// TwinCAT 3 PLC project TcoData
// Title: TcoData
// Company: Vortex.Library
// ProjectVersion: 0.6.0.913
// ProgramVersion: 3.1.4023.0
// libraries:
//   Tc2_Standard, * (Beckhoff Automation GmbH)
//   Tc2_System, * (Beckhoff Automation GmbH)
//   Tc3_Module, * (Beckhoff Automation GmbH)
//   TcoCore, 0.6.0.913 (Vortex.Library)
// project tree:
//   / PlcTask.TcTTO
//   POUs/Data/ TcoEntity.TcDUT, ITcoCrud.TcIO, TcoDataExchange.TcPOU, TcoDataTask.TcPOU, TcoExistsTask.TcPOU
//   POUs/ MAIN.TcPOU, MainContext.TcPOU
// real-time tasks:
//   TASK PlcTask: cycle T#10ms, priority 20, ADS port 350

CONFIGURATION TcoData
    RESOURCE PLC ON TwinCAT3
        TASK PlcTask(INTERVAL := T#10ms, PRIORITY := 20);
        PROGRAM MAIN WITH PlcTask : MAIN;
    END_RESOURCE
END_CONFIGURATION

// ---- POUs/Data/TcoEntity.TcDUT
(*~
    <docu>
        <summary>
            Base strucure of any data entity used in TcoDataExchange.
            <remarks>
                   <note type="information">
                    Inxton is required for this feature to work.
                   </note>
            </remarks>
        </summary>

        <example>
            [!code-pas[Declarations](~/../TcOpen/src/TcoData/src/XAE/XAE/TcoDataTests/POUs/Examples/SandboxData.TcDUT?name=SandboxData)]
        </example>
    </docu>
~*)
TYPE TcoEntity EXTENDS TcoCore.TcoStruct :
STRUCT
    {attribute wpf [Container(Layout.Stack)]}
    {attribute addProperty Name "<#ID#>"}
    {attribute clr [RenderIgnore("Control", "ShadowControl", "ControlSlim", "ShadowControlSlim")]}
    _EntityId : STRING(254);
END_STRUCT
END_TYPE

// ---- POUs/Data/ITcoCrud.TcIO
INTERFACE ITcoCrud

METHOD Create : TcoCore.ITcoTaskStatus
VAR_INPUT
	Identifier : STRING(255);
END_VAR
END_METHOD

METHOD Delete : TcoCore.ITcoTaskStatus
VAR_INPUT
	Identifier : STRING(255);
END_VAR
END_METHOD

METHOD Read : TcoCore.ITcoTaskStatus
VAR_INPUT
	Identifier : STRING(255);
END_VAR
END_METHOD

METHOD Update : TcoCore.ITcoTaskStatus
VAR_INPUT
	Identifier : STRING(255);
END_VAR
END_METHOD

END_INTERFACE

// ---- POUs/MAIN.TcPOU
PROGRAM INTERNAL MAIN
VAR
    Context : MainContext;
END_VAR

END_PROGRAM

// ---- POUs/MainContext.TcPOU
FUNCTION_BLOCK INTERNAL MainContext EXTENDS TcoCore.TcoContext
VAR
    fbProcessDataManger : TcoDataExchange(THIS^);
    test : TcoEntity;
END_VAR

(*~
    <docu>
        <summary>
            Main method of the TcoContext. This is the entry point of any control logic that belongs to this context.
            The call of this method is ensured by calling the <c>InstanceName.Run()</c> method, and it must not be called explicitly.
            This method is abstract, and it must be overridden in derived block.
        </summary>
    </docu>
~*)
METHOD PROTECTED Main
END_METHOD

END_FUNCTION_BLOCK

// ---- POUs/Data/TcoDataExchange.TcPOU
(*~
    <docu>
        <summary>
            Provides a mechanism to exchange data between PLC and an arbitrary data repository.
            TcoDataExchange support Create, Read, Update, Delete (CRUD) operations and some additional
            functions.
            TcoDataExchange **operates by convention on data member named `_data`** declared in the function block.
            The `_data` member must be of type that extends `TcoData.TcoEntity`.
            TcoDataEchange must be then inizialized in the higher level application where the repository
            and remote data exchange is configured.
            <remarks>
                   <note type="information">
                    Inxton is required for this feature to work.
                   </note>
            </remarks>
        </summary>

        <example>
            [!code-pas[Declarations](~/../TcOpen/src/TcoData/src/XAE/XAE/TcoDataTests/POUs/Examples/TcoDataManager.TcPOU?name=DataManagerDeclarations)]
            [!code-pas[SuperCall](~/../TcOpen/src/TcoData/src/XAE/XAE/TcoDataTests/POUs/Examples/TcoDataManager.TcPOU?name=DataManagerSuperCall)]
            [!code-pas[Data](~/../TcOpen/src/TcoData/src/XAE/XAE/TcoDataTests/POUs/Examples/SandboxData.TcDUT?name=SandboxData)]
            [!code-csharp[Main](~/../TcOpen/src/TcoData/tests/TcoDataExamples.Tests/SandboxContextTests.cs?name=RepositoryInitialization)]
        </example>
    </docu>
~*)
FUNCTION_BLOCK TcoDataExchange EXTENDS TcoCore.TcoObject IMPLEMENTS ITcoCrud
VAR
    (*~
        <docu>
            <summary>
                Instance of task that `creates` the entry into repository.
            </summary>
        </docu>
    ~*)
    _createTask : TcoDataTask(THIS^);
    (*~
        <docu>
            <summary>
                Instance of task that `reads` the entry from repository.
            </summary>
        </docu>
    ~*)
    _readTask : TcoDataTask(THIS^);
    (*~
        <docu>
            <summary>
                Instance of task that `updates` record in the repository.
            </summary>
        </docu>
    ~*)
    _updateTask : TcoDataTask(THIS^);
    (*~
        <docu>
            <summary>
                Instance of task that `deletes` record from the repository.
            </summary>
        </docu>
    ~*)
    _deleteTask : TcoDataTask(THIS^);
    (*~
        <docu>
            <summary>
                Instance of task that `check for existence` of a record with an `id` in the repository.
            </summary>
        </docu>
    ~*)
    _idExistsTask : TcoExistsTask(THIS^);
    (*~
        <docu>
            <summary>
                Instance of task that `creates inexisting or updates existing` record in the repository.
            </summary>
        </docu>
    ~*)
    _createOrUpdateTask : TcoDataTask(THIS^);
END_VAR

_createTask();
_readTask();
_updateTask();
_deleteTask();
_idExistsTask();
_createOrUpdateTask();

(*~
    <docu>
        <summary>
            Creates new entry in the Repository from `_data` member of this `TcoDataExchange`.
            <remarks>
                   <note type="information">
                    Inxton is required for this feature to work.
                   </note>
            </remarks>
        </summary>

        <example>
            [!code-pas[Main](~/../TcOpen/src/TcoData/src/XAE/XAE/TcoDataTests/POUs/Examples/SandboxContext.TcPOU?name=CreateCodeExample)]
        </example>
    </docu>
~*)
METHOD Create : TcoCore.ITcoTaskStatus
VAR_INPUT
    (*~
    <docu>
        <summary>
            Identifier of the data entry to be created in the repository.
        </summary>

    </docu>
    ~*)
    Identifier : STRING(255);
END_VAR
Create := _createTask.WithId(Identifier).Invoke();
THIS^.Messenger.Build().Append('<#Creating data item with id:#> ').Append(Identifier).As().AsTrace();
END_METHOD

(*~
    <docu>
        <summary>
            Creates or updates new entry in the Repository from `_data` member of this `TcoDataExchange`.
            <remarks>
                   <note type="information">
                    Inxton is required for this feature to work.
                   </note>
            </remarks>
        </summary>

        <example>
            [!code-pas[Main](~/../TcOpen/src/TcoData/src/XAE/XAE/TcoDataTests/POUs/Examples/SandboxContext.TcPOU?name=CreateOrUpdateCodeExample)]
        </example>
    </docu>
~*)
METHOD CreateOrUpdate : TcoCore.ITcoTaskStatus
VAR_INPUT
    (*~
        <docu>
            <summary>
                Identifier of the data entry to be created or updated in the repository.
            </summary>

        </docu>
    ~*)
    Identifier : STRING(255);
END_VAR
CreateOrUpdate := _createOrUpdateTask.WithId(Identifier).Invoke();
THIS^.Messenger.Build().Append('<#Creating or updating data item with id:#> ').Append(Identifier).As().AsTrace();
END_METHOD

(*~
    <docu>
        <summary>
            Deletes an item from the repository.
            <remarks>
                   <note type="information">
                    Inxton is required for this feature to work.
                   </note>
            </remarks>
        </summary>

        <example>
            [!code-pas[Main](~/../TcOpen/src/TcoData/src/XAE/XAE/TcoDataTests/POUs/Examples/SandboxContext.TcPOU?name=DeleteCodeExample)]
        </example>
    </docu>
~*)
METHOD Delete : TcoCore.ITcoTaskStatus
VAR_INPUT
    (*~
        <docu>
            <summary>
                Identifier of the data entry to be deleted from the repository.
            </summary>

        </docu>
    ~*)
    Identifier : STRING(255);
END_VAR
Delete := _deleteTask.WithId(Identifier).Invoke();
THIS^.Messenger.Build().Append('<#Deleting data item with id:#> ').Append(Identifier).As().AsTrace();
END_METHOD

(*~
    <docu>
        <summary>
            Determines if the entry with given `Identifier` exists in the repository.
            <remarks>
                   <note type="information">
                    Inxton is required for this feature to work.
                   </note>
            </remarks>
        </summary>

        <example>
            [!code-pas[Main](~/../TcOpen/src/TcoData/src/XAE/XAE/TcoDataTests/POUs/Examples/SandboxContext.TcPOU?name=ExistsCodeExample)]
        </example>
    </docu>
~*)
METHOD Exists : REFERENCE TO TcoExistsTask
VAR_INPUT
    (*~
        <docu>
            <summary>
                Identifier of the data entry for which the existence is to be checked.
            </summary>
        </docu>
    ~*)
    Identifier : STRING(255);
END_VAR
_idExistsTask.WithId(Identifier).Invoke();
THIS^.Messenger.Build().Append('<#Checking existence of data item with id:#> ').Append(Identifier).As().AsTrace();
Exists REF= _idExistsTask;
END_METHOD

METHOD FB_init : BOOL
VAR_INPUT
    bInitRetains : BOOL; // if TRUE, the retain variables are initialized (warm start / cold start)
    bInCopyCode : BOOL; // if TRUE, the instance afterwards gets moved into the copy code (online change)
    ParentObject : TcoCore.ITcoObject;
END_VAR
END_METHOD

(*~
    <docu>
        <summary>
            Reads data from the repository and stores it into `_data` member of this instance of `TcoDataExchange`.
            <remarks>
                   <note type="information">
                    Inxton is required for this feature to work.
                   </note>
            </remarks>
        </summary>

        <example>
            [!code-pas[Main](~/../TcOpen/src/TcoData/src/XAE/XAE/TcoDataTests/POUs/Examples/SandboxContext.TcPOU?name=ReadCodeExample)]
        </example>
    </docu>
~*)
METHOD Read : TcoCore.ITcoTaskStatus
VAR_INPUT
    (*~
        <docu>
            <summary>
                Identifier of the data entry to be retrieved from the repoository.
            </summary>
        </docu>
    ~*)
    Identifier : STRING(255);
END_VAR
Read := _readTask.WithId(Identifier).Invoke();
THIS^.Messenger.Build().Append('<#Reading data item with id:#> ').Append(Identifier).As().AsTrace();
END_METHOD

METHOD Restore : BOOL
VAR_INPUT
END_VAR
_createTask.Restore();
_readTask.Restore();
_updateTask.Restore();
_deleteTask.Restore();
_idExistsTask.Restore();
_createOrUpdateTask.Restore();
END_METHOD

(*~
    <docu>
        <summary>
            Updates data in the repository from `_data` member of this instance of `TcoDataExchange`.
            <remarks>
                   <note type="information">
                    Inxton is required for this feature to work.
                   </note>
            </remarks>
        </summary>

        <example>
            [!code-pas[Main](~/../TcOpen/src/TcoData/src/XAE/XAE/TcoDataTests/POUs/Examples/SandboxContext.TcPOU?name=UpdateCodeExample)]
        </example>
    </docu>
~*)
METHOD Update : TcoCore.ITcoTaskStatus
VAR_INPUT
    (*~
        <docu>
            <summary>
                Identifier of the data entry to be updated.
            </summary>
        </docu>
    ~*)
    Identifier : STRING(255);
END_VAR
Update := _updateTask.WithId(Identifier).Invoke();
THIS^.Messenger.Build().Append('<#Updating data item with id:#> ').Append(Identifier).As().AsTrace();
END_METHOD

END_FUNCTION_BLOCK

// ---- POUs/Data/TcoDataTask.TcPOU
(*~
    <docu>
        <summary>
            Data task is a remote task  <see cref="PlcDocu.TcoCore.RemoteTask"/> with a paramater.
        </summary>
        <param name="_identifier">The Identifier, ID  of an entity on which a CRUD operation should be executed</param>
        <remarks>Inxton is required for this feature to work</remarks>
    </docu>
~*)
FUNCTION_BLOCK TcoDataTask EXTENDS TcoCore.TcoRemoteTask
VAR
    (*~
    <docu>
        <summary>
            The Identifier, ID  of an entity on which a CRUD operation should be executed.
        </summary>
    </docu>
    ~*)
    _identifier : STRING(255);
END_VAR

SUPER^();

METHOD PUBLIC FB_init : BOOL
VAR_INPUT
    bInitRetains : BOOL; // if TRUE, the retain variables are initialized (warm start / cold start)
    bInCopyCode : BOOL; // if TRUE, the instance afterwards gets moved into the copy code (online change)
    ParentObject : TcoCore.ITcoObject;
END_VAR
END_METHOD

(*~
    <docu>
        <summary>
            Executes CRUD operation on data entry with given identifier.
        </summary>
        <remarks>Inxton is required for this feature to work</remarks>
    </docu>
~*)
METHOD WithId : REFERENCE TO TcoDataTask
VAR_INPUT
    (*~
    <docu>
        <summary>
            The Identifier, ID  of an entity on which a CRUD operation should be executed.
        </summary>
    </docu>
    ~*)
    inIdentifier : STRING(254);
END_VAR
THIS^._identifier := inIdentifier;
WithId REF= THIS^;
END_METHOD

END_FUNCTION_BLOCK

// ---- POUs/Data/TcoExistsTask.TcPOU
FUNCTION_BLOCK TcoExistsTask EXTENDS TcoDataTask
VAR
    _exists : BOOL;
END_VAR

SUPER^();

{attribute 'monitoring' := 'variable'}
PROPERTY Exists : BOOL
GET
Exists := _exists;
END_GET
END_PROPERTY

END_FUNCTION_BLOCK
